TYPE ST_HandShake_TrayMovement :
STRUCT

	
	
END_STRUCT
END_TYPE

(* stored: Version 1.1.0.1, ProductVersion 3.1.4024.12
   DUT ST_HandShake_TrayMovement: Id {25a240f0-167e-4a3e-8349-775bd7e34f45} *)
